DATA_BLOCK "Logica_PW_DB"
{ S7_Optimized_Access := 'TRUE' }
VERSION : 0.1
NON_RETAIN
"Logica_PW"

BEGIN

END_DATA_BLOCK

